// TwinCAT 3 PLC project ph_lv2_Communication_HTTP_REST
// Title: tclib_ph_lv2_http_rest
// Company: Poh
// Author: Poh
// ProjectVersion: 0.1.1.0
// ProgramVersion: 3.1.4020.1
// libraries:
//   Tc2_Standard, * (Beckhoff Automation GmbH)
//   Tc2_System, * (Beckhoff Automation GmbH)
//   tclib_ph_lv0, * (Poh)
//   tclib_ph_lv1_generic_communication_interface, * (Poh)
// project tree:
//   Lv2_Communication_REST_HTTP/Class Component/ C_HTTP_BASE.TcPOU, C_HTTP_HEADER.TcPOU, C_HTTP_VERSION.TcPOU
//   Lv2_Communication_REST_HTTP/ C_RESTFUL_CLIENT.TcPOU
//   Lv2_Communication_REST_HTTP/Datatype/ E_HTTP_RESPONSE_CODE.TcDUT, E_HTTP_STANDARD_HEADERS.TcDUT, E_HTTP_VERBS.TcDUT, LV2_HTTP_DATA_DEFINITIONS.TcGVL, T_HTTPSTRING.TcDUT (not stored)
//   Lv2_Communication_REST_HTTP/Http Message/ C_HTTP_REQUEST.TcPOU, C_HTTP_RESPONSE.TcPOU
//   Version/ Global_Version.TcGVL
// (motion and I/O tree: see PLC project ph_lv0)
// real-time tasks:
//   TASK PlcTask: cycle T#10ms, priority 20, ADS port 350
// variable links:

// ---- Lv2_Communication_REST_HTTP/Datatype/E_HTTP_RESPONSE_CODE.TcDUT
{attribute 'qualified_only'}
{attribute 'strict'}
TYPE E_HTTP_RESPONSE_CODE :
(
	//1xx : INFOMATIONAL
		HTTP_CONTINUE						:= 100,
		HTTP_SWITCH_PROTOCOL				:= 101,
	//2xx : SUCCESSFUL
		HTTP_OK 							:= 200,
		HTTP_CREATED 						:= 201,
		HTTP_ACCEPTED						:= 202,
		HTTP_NON_AUTHORITATIVE_INFORMATION	:= 203,
		HTTP_NO_CONTENT						:= 204,
		HTTP_RESET_CONTENT					:= 205,
		HTTP_PARTIAL_CONTENT				:= 206,
	//3xx : REDIRECTION
		HTTP_MULTIPLE_CHOICE				:= 300, //Link list. Max 5.
		HTTP_MOVED_PERMANENTLY				:= 301,
		HTTP_FOUND							:= 302,
		HTTP_SEE_OTHER						:= 303,
		HTTP_NOT_MODIFIED					:= 304,
		HTTP_USE_PROXY						:= 305,
		HTTP_UNUSED							:= 306,
		HTTP_TEMPORARY_REDIRECT				:= 307,
	//4xx : CLIENT ERROR
		HTTP_BAD_REQUEST 					:= 400,
		HTTP_UNAUTHORIZED 					:= 401,
		HTTP_PAYMENT_REQUIRED				:= 402,
		HTTP_FORBIDDEN 						:= 403,
		HTTP_NOT_FOUND 						:= 404,
		HTTP_METHOD_NOT_ALLOWED				:= 405,
		HTTP_NOT_ACCEPTABLE					:= 406,
		HTTP_PROXY_AUTHENTICATION_REQUIRED	:= 407,
		HTTP_REQUEST_TIMEOUT				:= 408,
		HTTP_CONFLICT						:= 409,
		HTTP_GONE							:= 410,
		HTTP_LENGTH_REQUIRED				:= 411,
		HTTP_PRECONDITION_FAILED			:= 412,
		HTTP_REQUEST_ENTITY_TOO_LARGE		:= 413,
		HTTP_REQUEST_URL_TOO_LONG			:= 414,
		HTTP_UNSUPPORTED_MEDIA_TYPE			:= 415,
		HTTP_REQUESTED_RANGE_NOT_SATISFIABLE:= 416,
		HTTP_EXPECTATION_FAILED				:= 417,
	//5xx : SERVER ERROR
		HTTP_INTERNAL_SERVER_ERROR 			:= 500,
		HTTP_NOT_IMPLEMENTED	 			:= 501,
		HTTP_BAD_GATEWAY		 			:= 502,
		HTTP_SERVICE_UNAVAILABLE 			:= 503,
		HTTP_GATEWAY_TIMEOUT	 			:= 504,
		HTTP_VERSION_NOT_SUPPORTED			:= 505
)UDINT;
END_TYPE

// ---- Lv2_Communication_REST_HTTP/Datatype/E_HTTP_STANDARD_HEADERS.TcDUT
{attribute 'qualified_only'}
{attribute 'strict'}
TYPE E_HTTP_STANDARD_HEADERS :
(
	//Request
		Accept_Charset_Header := 0,
		Accept_Encoding_Header,
		Accept_Language_Header,
		Authorization_Header,
		Expect_Header,
		From_Header,
		Host_Header,
		If_Match_Header,
		If_Modified_Since_Header,
		If_None_Match_Header,
		If_Range_Header,
		If_Unmodified_Since_Header,
		Max_Forwards_Header,
		Proxy_Authorization_Header,
		Range_Header,
		Referer_Header,
		Te_Header,
		User_Agent_Header,
	//Response
		Accept_Ranges_Header_Header,
		Age_Header_Header,
		ETag_Header,
		Location_Header,
		Proxy_Authenticate_Header,
		Retry_After_Header,
		Server_Header,
		Vary_Header,
		WWW_Authenticate_Header,
	Standard_Headers_Size
)UDINT;
END_TYPE

// ---- Lv2_Communication_REST_HTTP/Datatype/E_HTTP_VERBS.TcDUT
{attribute 'qualified_only'}
{attribute 'strict'}
TYPE E_HTTP_VERBS :
(
	//USED FOR RETRIEVING INFORMATION
		GET := 0,
	//SAME AS GET, BUT TRANSFERS THE STATUS LINE AND HEADER SECTION ONLY
		HEAD,
	//USED FOR SENDING DATA TO SERVER SUCH AS FILE UPLOAD, CUSTOMER INFO
		POST,
	//REPLACES ALL CURRENT REPRESENTATIONS OF TARGET RESOURCE WITH THE UPLOADED CONTENT
		PUT,
	//REMOVE ALL CURRENT REPRESENTATION OF TARGET RESOURCE GIVEN BY THE URI
		DELETE,
	//ESTABLISH A TUNNEL TO THE SERVER IDENTIFIED BY THE URL
		CONNECT,
	//DESCRIBE THE COMMUNICATION OPTIONS FOR TARGET RESOURCE
		OPTIONS,
	//PERFORMS A MESSAGE LOOP BACK TEST ALONG WITH THE PATH TO THE TARGET RESOURCE
		TRACE,
	VERB_COUNT
);
END_TYPE

// ---- Lv2_Communication_REST_HTTP/Datatype/LV2_HTTP_DATA_DEFINITIONS.TcGVL
{attribute 'qualified_only'}
VAR_GLOBAL CONSTANT
	//1xx : INFOMATIONAL
		HTTP_CONTINUE						: UDINT := 100;
		HTTP_SWITCH_PROTOCOL				: UDINT := 101;
	//2xx : SUCCESSFUL
		HTTP_OK 							: UDINT := 200;
		HTTP_CREATED 						: UDINT := 201;
		HTTP_ACCEPTED						: UDINT := 202;
		HTTP_NON_AUTHORITATIVE_INFORMATION	: UDINT := 203;
		HTTP_NO_CONTENT						: UDINT := 204;
		HTTP_RESET_CONTENT					: UDINT := 205;
		HTTP_PARTIAL_CONTENT				: UDINT := 206;
	//3xx : REDIRECTION
		HTTP_MULTIPLE_CHOICE				: UDINT := 300; //Link list. Max 5.
		HTTP_MOVED_PERMANENTLY				: UDINT := 301;
		HTTP_FOUND							: UDINT := 302;
		HTTP_SEE_OTHER						: UDINT := 303;
		HTTP_NOT_MODIFIED					: UDINT := 304;
		HTTP_USE_PROXY						: UDINT := 305;
		HTTP_UNUSED							: UDINT := 306;
		HTTP_TEMPORARY_REDIRECT				: UDINT := 307;
	//4xx : CLIENT ERROR
		HTTP_BAD_REQUEST 					: UDINT := 400;
		HTTP_UNAUTHORIZED 					: UDINT := 401;
		HTTP_PAYMENT_REQUIRED				: UDINT := 402;
		HTTP_FORBIDDEN 						: UDINT := 403;
		HTTP_NOT_FOUND 						: UDINT := 404;
		HTTP_METHOD_NOT_ALLOWED				: UDINT := 405;
		HTTP_NOT_ACCEPTABLE					: UDINT := 406;
		HTTP_PROXY_AUTHENTICATION_REQUIRED	: UDINT := 407;
		HTTP_REQUEST_TIMEOUT				: UDINT := 408;
		HTTP_CONFLICT						: UDINT := 409;
		HTTP_GONE							: UDINT := 410;
		HTTP_LENGTH_REQUIRED				: UDINT := 411;
		HTTP_PRECONDITION_FAILED			: UDINT := 412;
		HTTP_REQUEST_ENTITY_TOO_LARGE		: UDINT := 413;
		HTTP_REQUEST_URL_TOO_LONG			: UDINT := 414;
		HTTP_UNSUPPORTED_MEDIA_TYPE			: UDINT := 415;
		HTTP_REQUESTED_RANGE_NOT_SATISFIABLE: UDINT := 416;
		HTTP_EXPECTATION_FAILED				: UDINT := 417;
	//5xx : SERVER ERROR
		HTTP_INTERNAL_SERVER_ERROR 			: UDINT := 500;
		HTTP_NOT_IMPLEMENTED	 			: UDINT := 501;
		HTTP_BAD_GATEWAY		 			: UDINT := 502;
		HTTP_SERVICE_UNAVAILABLE 			: UDINT := 503;
		HTTP_GATEWAY_TIMEOUT	 			: UDINT := 504;
		HTTP_VERSION_NOT_SUPPORTED			: UDINT := 505;
	HTTP_VERB_STRING			: ARRAY[0..E_HTTP_VERBS.VERB_COUNT] OF STRING(15) := 
		[
			'GET',
			'HEAD',
			'PUT',
			'DELETE',
			'CONNECT',
			'OPTIONS',
			'TRACE',
			'_reserved_'
		];
	HTTP_STANDARD_HEADER_STRING : ARRAY[0..E_HTTP_STANDARD_HEADERS.Standard_Headers_Size] OF STRING(255) :=
		[
			'Accept-Charset',
			'Accept-Encoding',
			'Accept-Language',
			'Authorization',
			'Expect',
			'From',
			'Host',
			'If-Match',
			'If-Modified-Since',
			'If-None-Match',
			'If-Range',
			'If-Unmodified-Since',
			'Max-Forwards',
			'Proxy-Authorization',
			'Range',
			'Referer',
			'TE',
			'User-Agent',
			'Accept-Ranges',
			'Age',
			'ETag',
			'Location',
			'Proxy-Authenticate',
			'Retry-After',
			'Server',
			'Vary',
			'WWW-Authenticate',
			'_reserved_'
		];
END_VAR

// ---- Version/Global_Version.TcGVL
{attribute 'TcGenerated'}
// This function has been automatically generated from the project information.
VAR_GLOBAL CONSTANT
	{attribute 'const_non_replaced'}
	{attribute 'linkalways'}
	stLibVersion_tclib_ph_lv2_http_rest : ST_LibVersion := (iMajor := 0, iMinor := 1, iBuild := 1, iRevision := 0, sVersion := '0.1.1.0');
END_VAR

// ---- Lv2_Communication_REST_HTTP/Class Component/C_HTTP_BASE.TcPOU
FUNCTION_BLOCK C_HTTP_BASE
VAR_INPUT
END_VAR
VAR_OUTPUT
END_VAR
VAR
END_VAR

PROPERTY Header_Delimiter : STRING(2)
GET
Header_Delimiter := ': ';
END_GET
END_PROPERTY

PROPERTY Line_Space : String(1)
GET
Line_Space := ' ';
END_GET
END_PROPERTY

PROPERTY Line_Terminator : STRING(2)
GET
Line_Terminator := '$R$N';
END_GET
END_PROPERTY

PROPERTY PROTECTED Url_Split_Charactor : STRING(1)
GET
Url_Split_Charactor := '/';
END_GET
END_PROPERTY

END_FUNCTION_BLOCK

// ---- Lv2_Communication_REST_HTTP/Class Component/C_HTTP_HEADER.TcPOU
FUNCTION_BLOCK C_HTTP_HEADER EXTENDS C_HTTP_BASE
VAR_INPUT
END_VAR
VAR_OUTPUT
END_VAR
VAR
	_FieldName 	: STRING(255);
	_HeaderField: STRING(255);
END_VAR

METHOD Equals : BOOL
VAR_INPUT
	IN_HEADER : POINTER TO C_HTTP_HEADER;
END_VAR
VAR
	_stringInternal 	: STRING(255);
	_stringInput 		: STRING(255);
	_lenString			: INT;
	_i 					: DINT;
END_VAR
IF LEN(IN_HEADER^.Field_Name) <> LEN(THIS^.Field_Name) THEN
	Equals := FALSE;
ELSIF LEN(IN_HEADER^.Header_Field) <> LEN(THIS^.Header_Field) THEN
	Equals := FALSE;
ELSE
	_stringInternal := THIS^.Field_Name;
	_stringInput := IN_HEADER^.Field_Name;
	_lenString := LEN(_stringInternal);
	_i := MEMCMP(ADR(_stringinternal),ADR(_stringInput), _lenString);
	IF _i <> 0 THEN
		Equals := FALSE;
	ELSE
		_stringInternal := THIS^.Header_Field;
		_stringInput := IN_HEADER^.Header_Field;
		_lenString := LEN(_stringInternal);
		_i := MEMCMP(ADR(_stringinternal),ADR(_stringInput), _lenString);
		IF _i <> 0 THEN
			Equals := FALSE;
		ELSE
			Equals := TRUE;
		END_IF
	END_IF
END_IF
END_METHOD

METHOD FB_init : BOOL
VAR_INPUT
	bInitRetains : BOOL; // if TRUE, the retain variables are initialized (warm start / cold start)
	bInCopyCode : BOOL;  // if TRUE, the instance afterwards gets moved into the copy code (online change)
	Name : STRING(255);
END_VAR
_FieldName := Name;
END_METHOD

PROPERTY Field_Name : STRING(255)
GET
Field_Name := _FieldName;
END_GET
SET
_FieldName := Field_Name;
END_SET
END_PROPERTY

PROPERTY Header_Field : STRING(255)
GET
Header_Field := _HeaderField;
END_GET
SET
_HeaderField := Header_Field;
END_SET
END_PROPERTY

METHOD Parse : RETURN_CODE
VAR_INPUT
	IN_STRING	: STRING(255);
END_VAR
VAR 
	_DELIMIT_POSITION : INT;
	_ENDLINE_POSITION : INT;
END_VAR
_DELIMIT_POSITION := FIND(IN_STRING, SUPER^.Header_Delimiter);
IF _DELIMIT_POSITION = 0 THEN
	Parse := ph_lv0.LV0_RETURNCODE.RETURN_ERROR + 1;
ELSE
	_ENDLINE_POSITION := FIND(IN_STRING, SUPER^.Line_Terminator);
	IF _ENDLINE_POSITION = 0 THEN
		Parse := ph_lv0.LV0_RETURNCODE.RETURN_ERROR + 2;
	ELSE
		_FieldName := MID(IN_STRING, _DELIMIT_POSITION - 1, 1);
		_HeaderField := MID(IN_STRING, _ENDLINE_POSITION - (_DELIMIT_POSITION + 2), _DELIMIT_POSITION + 2); 
		Parse := ph_lv0.LV0_RETURNCODE.RETURN_SUCCESS;
	END_IF
END_IF
END_METHOD

METHOD ToString : String(255)
VAR_INPUT
END_VAR
ToString := CONCAT(THIS^.Field_Name,
				CONCAT(SUPER^.Header_Delimiter, 
					CONCAT(THIS^.Header_Field,
						SUPER^.Line_Terminator
					)
				)
			);
END_METHOD

END_FUNCTION_BLOCK

// ---- Lv2_Communication_REST_HTTP/Class Component/C_HTTP_VERSION.TcPOU
FUNCTION_BLOCK C_HTTP_VERSION
VAR_INPUT
END_VAR
VAR_OUTPUT
END_VAR
VAR
	_Major : UINT := 1;
	_Minor : UINT := 0;
END_VAR

METHOD FB_init : BOOL
VAR_INPUT
	bInitRetains : BOOL; // if TRUE, the retain variables are initialized (warm start / cold start)
	bInCopyCode : BOOL;  // if TRUE, the instance afterwards gets moved into the copy code (online change)
	Major_Version : UINT;
	Minor_Version : UINT;
END_VAR
Major := Major_Version;
Minor := Minor_Version;
END_METHOD

PROPERTY Major : uint
GET
Major := _Major;
END_GET
SET
_Major := Major;
END_SET
END_PROPERTY

PROPERTY Minor : uint
GET
Minor := _Minor;
END_GET
SET
_Minor := Minor;
END_SET
END_PROPERTY

METHOD ToString : String(255)
VAR_INPUT
END_VAR
VAR
	_head 	: STRING(5) := 'HTML/';
END_VAR
ToString := CONCAT(_head, CONCAT(UINT_TO_STRING(_Major), CONCAT('.',UINT_TO_STRING(_Minor))));
END_METHOD

END_FUNCTION_BLOCK

// ---- Lv2_Communication_REST_HTTP/C_RESTFUL_CLIENT.TcPOU
FUNCTION_BLOCK C_RESTFUL_CLIENT
VAR_INPUT
END_VAR
VAR_OUTPUT
END_VAR
VAR
	_ifc_Communication 	: IFC_GENERIC_COMMUNICATION_INTERFACE;
	_c_HttpRequest		: C_HTTP_REQUEST;
END_VAR

END_FUNCTION_BLOCK

// ---- Lv2_Communication_REST_HTTP/Http Message/C_HTTP_REQUEST.TcPOU
FUNCTION_BLOCK C_HTTP_REQUEST EXTENDS C_HTTP_BASE
VAR_INPUT
END_VAR
VAR_OUTPUT
END_VAR
VAR
	_MethodRequest		: E_HTTP_VERBS;
	_Url				: STRING(255);	
	_c_HttpVersion 		: C_HTTP_VERSION(Major_Version:= 1, Minor_Version:= 1);
	
	_Header 			: ARRAY[0..15] OF C_HTTP_HEADER(Name:= '');
	
	_MessageBody		: T_HTTPSTRING;
END_VAR

METHOD PRIVATE Get_Headers : STRING(255)
VAR_INPUT
END_VAR
VAR 
	_m : INT := 0;
	_mn : INT := 15;
	_buffer : STRING(255) := '';
END_VAR
FOR _m := 0 TO _mn BY 1 DO
	_buffer := CONCAT(_buffer, THIS^._Header[_m].ToString());
END_FOR
Get_Headers := _buffer;
END_METHOD

METHOD PRIVATE Get_RequestLine : String(255)
VAR_INPUT
END_VAR
Get_RequestLine :=	CONCAT(LV2_HTTP_DATA_DEFINITIONS.HTTP_VERB_STRING[THIS^._MethodRequest],
						CONCAT(SUPER^.Line_Space, 
							CONCAT(_Url,
								CONCAT(SUPER^.Line_Space,
									CONCAT(_c_HttpVersion.ToString(),
										SUPER^.Line_Terminator
									)
								)
							)
						)
					);
END_METHOD

PROPERTY Major_Version : uint
GET
Major_Version := _c_HttpVersion.Major;;
END_GET
END_PROPERTY

PROPERTY Message_Body : STRING(255)
GET
Message_Body := _MessageBody;
END_GET
SET
_MessageBody := Message_Body;
END_SET
END_PROPERTY

PROPERTY Minor_Version : uint
GET
Minor_Version := _c_HttpVersion.Minor;
END_GET
END_PROPERTY

METHOD Parse : RETURN_CODE
VAR_INPUT
END_VAR
END_METHOD

METHOD ToString : STRING(255)
VAR_INPUT
END_VAR
ToString :=	CONCAT(THIS^.Get_RequestLine(),
				CONCAT(THIS^.Get_Headers(),
					CONCAT(SUPER^.Line_Terminator,
						THIS^.Message_Body
					)
				)
			);
END_METHOD

PROPERTY Url : String(255)
GET
Url := _url;
END_GET
SET
_url := url;
END_SET
END_PROPERTY

PROPERTY Verb : E_HTTP_VERBS
GET
Verb := _MethodRequest;
END_GET
SET
_MethodRequest := Verb;
END_SET
END_PROPERTY

END_FUNCTION_BLOCK

// ---- Lv2_Communication_REST_HTTP/Http Message/C_HTTP_RESPONSE.TcPOU
FUNCTION_BLOCK C_HTTP_RESPONSE EXTENDS C_HTTP_BASE
VAR_INPUT
END_VAR
VAR_OUTPUT
END_VAR
VAR
	_ResponseCode		: E_HTTP_RESPONSE_CODE;
	_Url				: STRING(255);	
	_c_HttpVersion 		: C_HTTP_VERSION(Major_Version:= 1, Minor_Version:= 1);
	
	_Header 			: ARRAY[0..15] OF C_HTTP_HEADER(Name:= '');
	
	_MessageBody		: T_HTTPSTRING;
END_VAR

PROPERTY Major_Version : uint
GET
Major_Version := _c_HttpVersion.Major;;
END_GET
END_PROPERTY

PROPERTY Minor_Version : uint
GET
Minor_Version := _c_HttpVersion.Minor;
END_GET
END_PROPERTY

END_FUNCTION_BLOCK
